SYSTEM Waterfilter_Backup
  (* Version 1.0, 2023-01-19, AK124017 *)
  APPLICATION Application
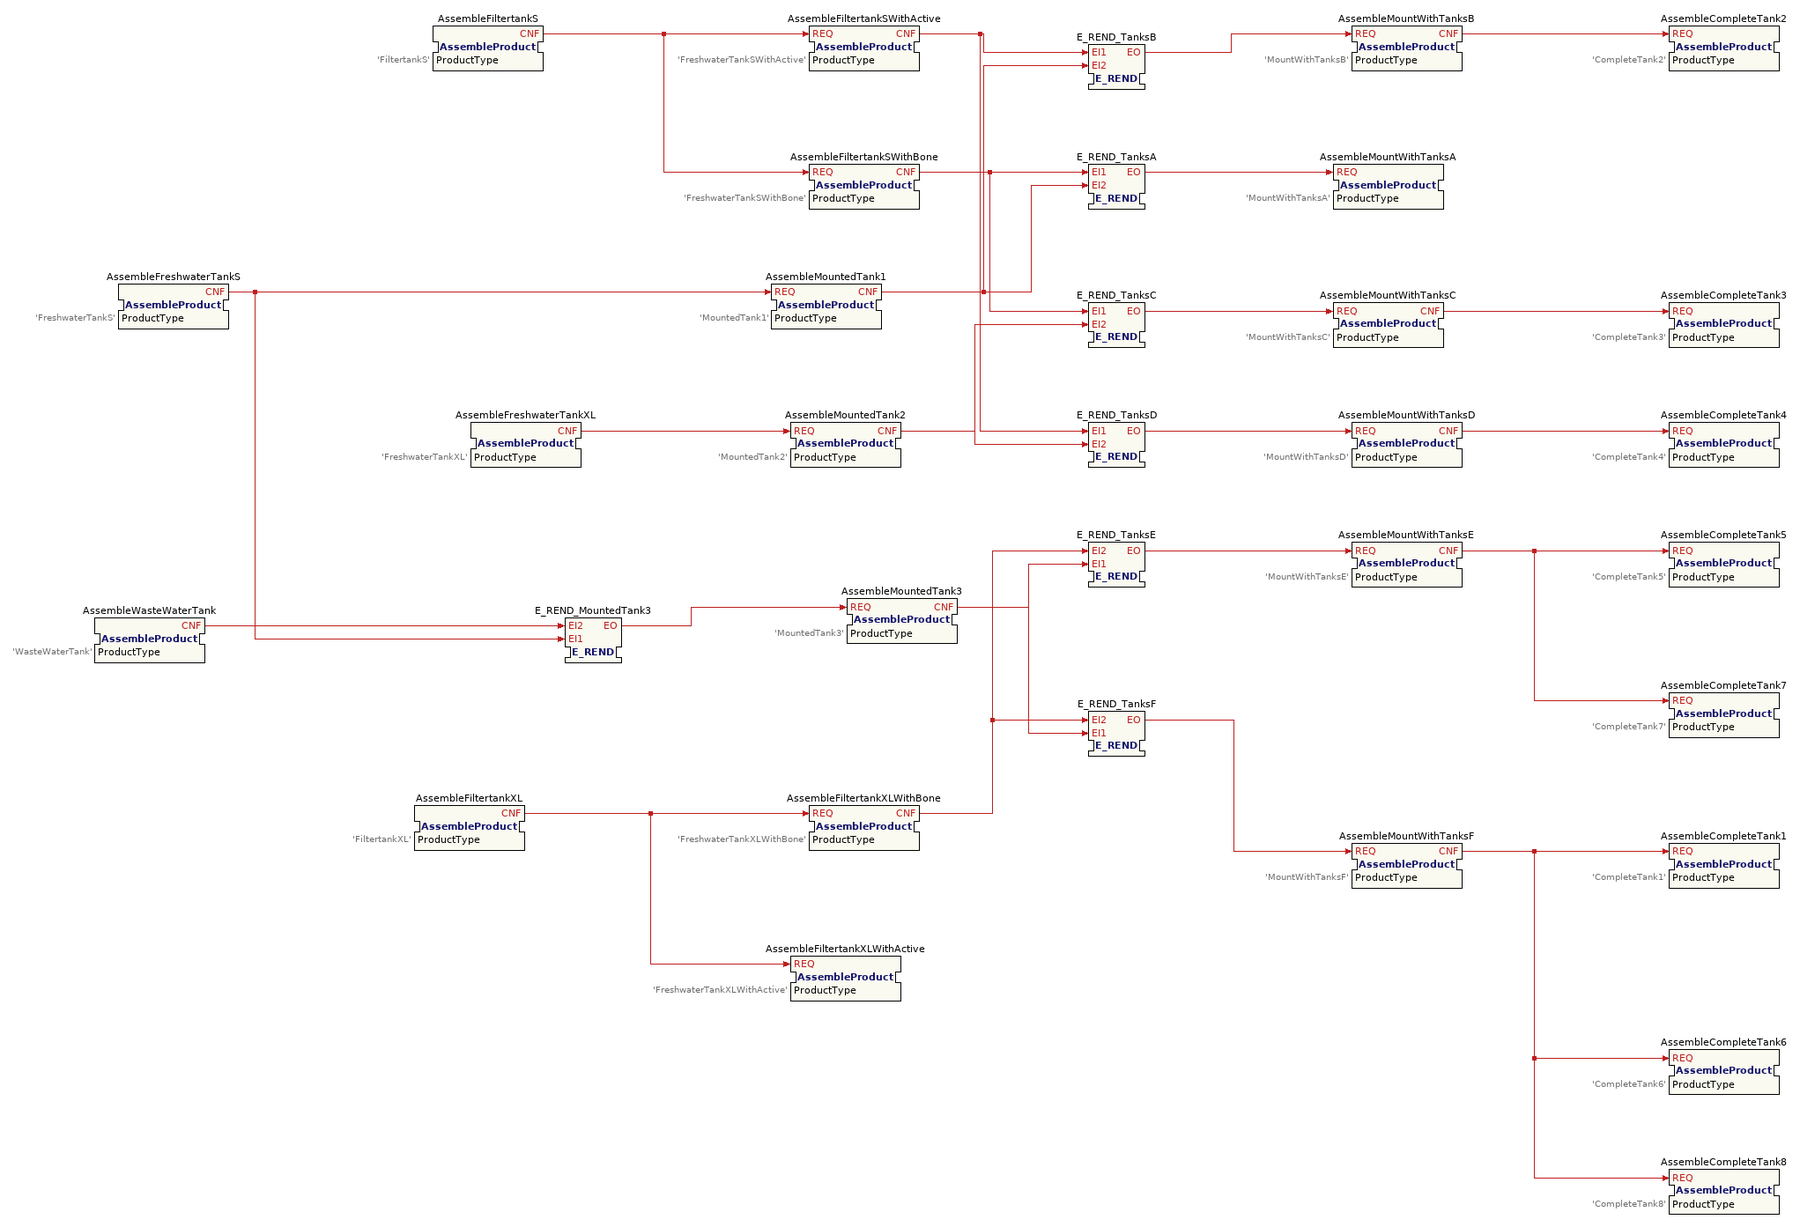
    FBS
      AssembleFiltertankS : AssembleProduct(ProductType := 'FiltertankS');
      AssembleFiltertankSWithActive : AssembleProduct(ProductType := 'FreshwaterTankSWithActive');
      AssembleFiltertankSWithBone : AssembleProduct(ProductType := 'FreshwaterTankSWithBone');
      AssembleMountWithTanksA : AssembleProduct(ProductType := 'MountWithTanksA');
      AssembleMountWithTanksE : AssembleProduct(ProductType := 'MountWithTanksE');
      AssembleMountWithTanksF : AssembleProduct(ProductType := 'MountWithTanksF');
      AssembleCompleteTank8 : AssembleProduct(ProductType := 'CompleteTank8');
      AssembleFiltertankXLWithBone : AssembleProduct(ProductType := 'FreshwaterTankXLWithBone');
      AssembleFiltertankXLWithActive : AssembleProduct(ProductType := 'FreshwaterTankXLWithActive');
      AssembleFiltertankXL : AssembleProduct(ProductType := 'FiltertankXL');
      E_REND_TanksA : E_REND;
      AssembleWasteWaterTank : AssembleProduct(ProductType := 'WasteWaterTank');
      AssembleFreshwaterTankS : AssembleProduct(ProductType := 'FreshwaterTankS');
      E_REND_MountedTank3 : E_REND;
      AssembleMountedTank3 : AssembleProduct(ProductType := 'MountedTank3');
      AssembleMountedTank1 : AssembleProduct(ProductType := 'MountedTank1');
      AssembleMountWithTanksB : AssembleProduct(ProductType := 'MountWithTanksB');
      E_REND_TanksB : E_REND;
      AssembleFreshwaterTankXL : AssembleProduct(ProductType := 'FreshwaterTankXL');
      AssembleMountedTank2 : AssembleProduct(ProductType := 'MountedTank2');
      E_REND_TanksC : E_REND;
      E_REND_TanksD : E_REND;
      AssembleMountWithTanksC : AssembleProduct(ProductType := 'MountWithTanksC');
      AssembleMountWithTanksD : AssembleProduct(ProductType := 'MountWithTanksD');
      E_REND_TanksF : E_REND;
      E_REND_TanksE : E_REND;
      AssembleCompleteTank1 : AssembleProduct(ProductType := 'CompleteTank1');
      AssembleCompleteTank2 : AssembleProduct(ProductType := 'CompleteTank2');
      AssembleCompleteTank3 : AssembleProduct(ProductType := 'CompleteTank3');
      AssembleCompleteTank4 : AssembleProduct(ProductType := 'CompleteTank4');
      AssembleCompleteTank5 : AssembleProduct(ProductType := 'CompleteTank5');
      AssembleCompleteTank6 : AssembleProduct(ProductType := 'CompleteTank6');
      AssembleCompleteTank7 : AssembleProduct(ProductType := 'CompleteTank7');
    END_FBS
    EVENT_CONNECTIONS
      AssembleFiltertankS.CNF TO AssembleFiltertankSWithActive.REQ;
      AssembleFiltertankS.CNF TO AssembleFiltertankSWithBone.REQ;
      AssembleFiltertankXL.CNF TO AssembleFiltertankXLWithBone.REQ;
      AssembleFiltertankSWithBone.CNF TO E_REND_TanksA.EI1;
      E_REND_TanksA.EO TO AssembleMountWithTanksA.REQ;
      AssembleWasteWaterTank.CNF TO E_REND_MountedTank3.EI2;
      AssembleFreshwaterTankS.CNF TO E_REND_MountedTank3.EI1;
      E_REND_MountedTank3.EO TO AssembleMountedTank3.REQ;
      AssembleFreshwaterTankS.CNF TO AssembleMountedTank1.REQ;
      AssembleFiltertankSWithActive.CNF TO E_REND_TanksB.EI1;
      E_REND_TanksB.EO TO AssembleMountWithTanksB.REQ;
      AssembleFreshwaterTankXL.CNF TO AssembleMountedTank2.REQ;
      AssembleFiltertankSWithBone.CNF TO E_REND_TanksC.EI1;
      AssembleFiltertankSWithActive.CNF TO E_REND_TanksD.EI1;
      AssembleMountedTank1.CNF TO E_REND_TanksB.EI2;
      AssembleMountedTank1.CNF TO E_REND_TanksA.EI2;
      AssembleMountedTank2.CNF TO E_REND_TanksC.EI2;
      AssembleMountedTank2.CNF TO E_REND_TanksD.EI2;
      E_REND_TanksD.EO TO AssembleMountWithTanksD.REQ;
      E_REND_TanksC.EO TO AssembleMountWithTanksC.REQ;
      AssembleFiltertankXL.CNF TO AssembleFiltertankXLWithActive.REQ;
      AssembleFiltertankXLWithBone.CNF TO E_REND_TanksE.EI2;
      AssembleFiltertankXLWithBone.CNF TO E_REND_TanksF.EI2;
      AssembleMountedTank3.CNF TO E_REND_TanksE.EI1;
      AssembleMountedTank3.CNF TO E_REND_TanksF.EI1;
      E_REND_TanksE.EO TO AssembleMountWithTanksE.REQ;
      E_REND_TanksF.EO TO AssembleMountWithTanksF.REQ;
      AssembleMountWithTanksF.CNF TO AssembleCompleteTank1.REQ;
      AssembleMountWithTanksB.CNF TO AssembleCompleteTank2.REQ;
      AssembleMountWithTanksC.CNF TO AssembleCompleteTank3.REQ;
      AssembleMountWithTanksD.CNF TO AssembleCompleteTank4.REQ;
      AssembleMountWithTanksE.CNF TO AssembleCompleteTank5.REQ;
      AssembleMountWithTanksF.CNF TO AssembleCompleteTank6.REQ;
      AssembleMountWithTanksE.CNF TO AssembleCompleteTank7.REQ;
      AssembleMountWithTanksF.CNF TO AssembleCompleteTank8.REQ;
    END_CONNECTIONS
  END_APPLICATION
END_SYSTEM
